FUNCTION_BLOCK FB_OffState IMPLEMENTS I_State
VAR_INPUT
END_VAR
VAR_OUTPUT
END_VAR
VAR
	pMachine : POINTER TO FB_StateMachine;
END_VAR

PROPERTY Description : STRING
GET
Description := 'Heat pump is switched off';
END_GET
END_PROPERTY

METHOD ErrorDetected : BOOL
VAR_INPUT
	errorEvents		: ST_ErrorEvents;
END_VAR
VAR
	message				: STRING(255);
END_VAR
END_METHOD

//FB_Init ist immer implizit verfügbar und wird primär für die Initialisierung verwendet.
//Der Rückgabewert wird nicht ausgewertet. Für gezielte Einflussnahme können Sie
//die Methoden explizit deklarieren und darin mit dem Standard-Initialisierungscode 
//zusätzlichen Code bereitstellen. Sie können den Rückgabewert auswerten.
METHOD FB_Init: BOOL
VAR_INPUT    
	bInitRetains: BOOL; // TRUE: Die Retain-Variablen werden initialisiert (Reset warm / Reset kalt)    
	bInCopyCode: BOOL;  // TRUE: Die Instanz wird danach in den Kopiercode kopiert (Online-Change)
	pMachine : POINTER TO FB_StateMachine;
END_VAR
THIS^.pMachine := pMachine;
END_METHOD

METHOD HeatIsRequested : BOOL
END_METHOD

METHOD LimitValuesAreExceeded : BOOL
END_METHOD

PROPERTY Name : STRING
GET
Name := 'Off';
END_GET
END_PROPERTY

PROPERTY State : E_State
GET
State := E_State.OFF;
END_GET
END_PROPERTY

METHOD TargetTemeperatureReached : BOOL
END_METHOD

METHOD UserPressedConfirmationButton : BOOL
END_METHOD

METHOD UserPressedSwitchOffButton : BOOL
END_METHOD

METHOD UserPressedSwitchOnButton : BOOL
ADSLOGSTR(ADSLOG_MSGTYPE_HINT, 'Einschalt Button wurde gedrückt -> %s', pMachine^.IdleState.Name);
pMachine^.SetState(pMachine^.IdleState);
END_METHOD

METHOD WaterHasCooledDown : BOOL
END_METHOD

END_FUNCTION_BLOCK

(* stored: Version 1.1.0.1
   POU FB_OffState: Id {81ed5e23-43bf-42e4-b314-a27a2acf9feb}, SpecialFunc None
   Property Description: Id {a23b52e3-14dd-4d1a-9c76-ef416d6f3d95}
   Get Get: Id {fdacbbeb-9f62-4ad4-8052-f6c5c3b7ba19}
   Method ErrorDetected: Id {1888cc77-ab19-429d-b5dc-9fd3ac4091b4}
   Method FB_init: Id {98bea1d9-064f-4e7b-bbff-5c1ffd972edc}
   Method HeatIsRequested: Id {bc849c3d-c10e-4743-b977-6435d1cdc9a1}
   Method LimitValuesAreExceeded: Id {5cac69aa-9a91-4532-8eb8-d799072b6f5b}
   Property Name: Id {2c52335e-5d4a-4ba6-8676-9c0b15fb0662}
   Get Get: Id {5bc9d40e-cee5-4ee4-823f-4fb0e1f3908a}
   Property State: Id {e9b35d77-403c-47b3-b5d5-c12b8407686e}
   Get Get: Id {5cf49127-fb9c-4307-a0b0-382199956e67}
   Method TargetTemeperatureReached: Id {03af484f-99f7-499a-bbd9-92b7758ce7e4}
   Method UserPressedConfirmationButton: Id {7c75e75b-3c89-4d24-b3fb-fe98e8a0d70e}
   Method UserPressedSwitchOffButton: Id {304776ef-1c80-4d97-a074-24b2a44303eb}
   Method UserPressedSwitchOnButton: Id {3e4c940e-09ad-46ae-a819-deeb3286e35e}
   Method WaterHasCooledDown: Id {df284c9a-4c2c-49fb-8cfb-cdf35d9d5fda} *)
